{attribute 'qualified_only'}
VAR_GLOBAL
		EtherCAT_Master_AMIxxxx : EtherCAT_Master_AMIxxxx_FECF87C2;
		EtherCAT_Master_APSxxxx : EtherCAT_Master_APSxxxx_6FACD001;
		EtherCAT_Master_ATxxxx : EtherCAT_Master_ATxxxx_83672136;
		EtherCAT_Master_AXxxxx : EtherCAT_Master_AXxxxx_5BD89A80;
		EtherCAT_Master_BKCUCX : EtherCAT_Master_BKCUCX_8F70BCEA;
		EtherCAT_Master_EJxxxx : EtherCAT_Master_EJxxxx_A1D13F1B;
		EtherCAT_Master_EKxxxx : EtherCAT_Master_EKxxxx_AFFC15C4;
		EtherCAT_Master_ELMxxxx : EtherCAT_Master_ELMxxxx_F3377F79;
		EtherCAT_Master_ELxxxx : EtherCAT_Master_ELxxxx_D51EE2EF;
		EtherCAT_Master_ELXxxxx : EtherCAT_Master_ELXxxxx_037A66B5;
		EtherCAT_Master_EMxxxx : EtherCAT_Master_EMxxxx_4F6AEAF3;
		EtherCAT_Master_EPPxxxx : EtherCAT_Master_EPPxxxx_7CC0E3EC;
		EtherCAT_Master_EPxxxx : EtherCAT_Master_EPxxxx_AD623DA0;
		EtherCAT_Master_EQxxxx : EtherCAT_Master_EQxxxx_C1E8A49A;
		EtherCAT_Master_ERxxxx : EtherCAT_Master_ERxxxx_D3400E61;
		EtherCAT_Master_KLxxxx : EtherCAT_Master_KLxxxx_4E9397D5;
		EtherCAT_Master_KLxxxx_1 : EtherCAT_Master_KLxxxx_1_B89C6D7A;
		EtherCAT_Master_KLxxxx_2 : EtherCAT_Master_KLxxxx_2_C1BBE75B;
		EtherCAT_Master_Duplicates : EtherCAT_Master_Duplicates_FF3295D1;
END_VAR

(* stored: Version 1.2.0.0, ProductVersion 3.1.4024.9
   GVL GVL_iXlinker: Id {ad1250ed-77f8-4b8c-9398-0ddad9706fc3} *)
